FUNCTION_BLOCK Render (* Function block to display and animate an Image *)
  (* Standard: 61499-2 *)
  (* Version 0.2, 2006-01-05, Anirudha, UoA, Added Layer attribute *)
  (* Version 0.1, 2005-12-04, Anirudha, UoA, Added Angle attribute *)
  (* Compiler header: package fb.rt.vhmi; *)
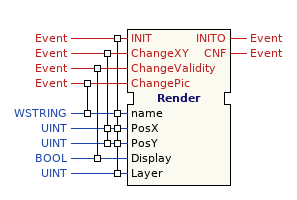
  EVENT_INPUT
    INIT WITH name, PosX, PosY, Layer; (* Initialization Request *)
    ChangeXY WITH PosX, PosY; (* Normal Execution Request *)
    ChangeValidity WITH Display;
    ChangePic WITH name;
  END_EVENT
  EVENT_OUTPUT
    INITO; (* Initialization Confirm *)
    CNF; (* Execution Confirmation *)
  END_EVENT
  VAR_INPUT
    name : WSTRING;
    PosX : UINT;
    PosY : UINT;
    Display : BOOL;
    Layer : UINT;
  END_VAR
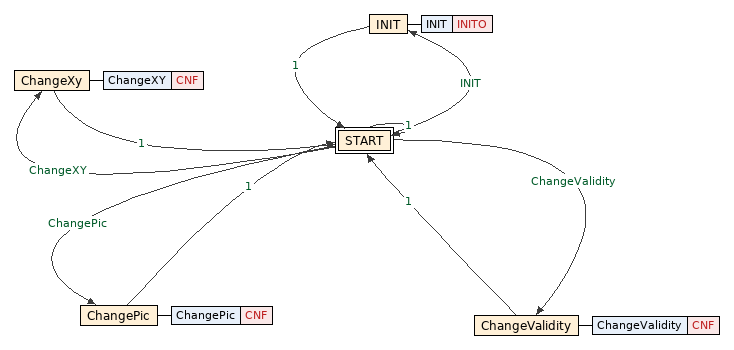
  EC_STATES
    START; (* Initial State *)
    INIT : INIT -> INITO; (* Initialization *)
    ChangeXy : ChangeXY -> CNF;
    ChangeValidity : ChangeValidity -> CNF;
    ChangePic : ChangePic -> CNF;
  END_STATES
  EC_TRANSITIONS
    START TO INIT := INIT;
    INIT TO START := 1;
    START TO ChangeXy := ChangeXY;
    START TO ChangeValidity := ChangeValidity;
    ChangeXy TO START := 1;
    ChangeValidity TO START := 1;
    START TO START := 1;
    START TO ChangePic := ChangePic;
    ChangePic TO START := 1;
  END_TRANSITIONS
  ALGORITHM INIT IN Java: (* Initialization algorithm *)
//System.out.print("Name: ");
//System.out.println(name.value);
//System.out.print("Position: ");
//System.out.print(PosX.value);
//System.out.print(",");
//System.out.print(PosY.value);
ID = ((ImageResource) this.resource).addImage(loadImage(name.value),PosX.value,PosY.value,Layer.value);
((ImageDev) this.getDevice()).frame.repaint();
//String abd = "I am " + name.value + " with ID " + ID;
//System.out.println(abd);
if (Display.value == false)
  service_ChangeValidity(true);
  END_ALGORITHM
  ALGORITHM ChangeXY IN Java:
((SampleFrame)((ImageDev)(this.getDevice())).frame).redrawXY(ID,PosX.value,PosY.value);
  END_ALGORITHM
  ALGORITHM ChangeValidity IN Java:
((SampleFrame)((ImageDev)(this.getDevice())).frame).setValidity(ID,Display.value);
  END_ALGORITHM
  ALGORITHM ChangePic IN Java:

  END_ALGORITHM
END_FUNCTION_BLOCK
